{attribute 'linkalways'} 
{attribute 'no_explicit_call' := 'This FB is a CLASS and must be accessed using methods or properties'}
{attribute 'enable_dynamic_creation'}
FUNCTION_BLOCK _ULINT EXTENDS NumericDatatypeBase
VAR
	localData : ULINT;
	activeData : REFERENCE TO ULINT REF= localData;
END_VAR

PROPERTY PUBLIC Address : PVOID
GET
Address := ADR(activeData);
END_GET
END_PROPERTY

METHOD PUBLIC ClearReference
VAR_INPUT
END_VAR
activeData REF= localData;
END_METHOD

METHOD PUBLIC Clone : I_Datatype
VAR
    pClone : POINTER TO _ULINT;
END_VAR
pClone := __NEW(_ULINT(InitialValue := Value));
Clone := pClone^;
END_METHOD

METHOD FB_init : BOOL
VAR_INPUT
	bInitRetains : BOOL; // if TRUE, the retain variables are initialized (warm start / cold start)
	bInCopyCode : BOOL;  // if TRUE, the instance afterwards gets moved into the copy code (online change)
	InitialValue : ULINT;
END_VAR
localData := InitialValue;
END_METHOD

PROPERTY PUBLIC IsFloat : BOOL
GET
IsFloat := FALSE;
END_GET
END_PROPERTY

PROPERTY PUBLIC IsSigned : BOOL
GET
IsSigned := FALSE;
END_GET
END_PROPERTY

PROPERTY PUBLIC LowerBound : ULINT
GET
LowerBound := DatatypeLimits.ULINT_LOWER_LIMIT;
END_GET
END_PROPERTY

METHOD PUBLIC MakeReferenceTo
VAR_INPUT
	ReferenceTarget : REFERENCE TO ULINT;
END_VAR
activeData REF= ReferenceTarget;
END_METHOD

METHOD PROTECTED SerializeLowerbound
VAR_INPUT
	Serializer : I_Serializer;
END_VAR
Serializer.AddUlint(Lowerbound);
END_METHOD

METHOD PROTECTED SerializeUpperbound
VAR_INPUT
	Serializer : I_Serializer;
END_VAR
Serializer.AddUlint(Upperbound);
END_METHOD

METHOD PUBLIC SerializeWith
VAR_INPUT
	Serializer : I_Serializer;
END_VAR
Serializer.AddUlint(activeData);
END_METHOD

PROPERTY PUBLIC Size : UDINT
GET
Size := SIZEOF(activeData);
END_GET
END_PROPERTY

METHOD TryDeserializeFrom : BOOL
VAR_INPUT
	Deserializer : I_Deserializer;
	Feedback : I_DeserializerFeedback;
END_VAR
TryDeserializeFrom := Deserializer.TryGetUlint(activeData, Feedback);
END_METHOD

METHOD TryMakeReferenceTo : BOOL
VAR_INPUT
	Target : I_Datatype;
END_VAR
VAR
	pTargetData : POINTER TO ULINT;
END_VAR
IF NOT (Target.TypeName = TypeName) THEN
	RETURN;
END_IF

pTargetData := Target.Address;
activeData REF= pTargetData^;
TryMakeReferenceTo := TRUE;
END_METHOD

PROPERTY PUBLIC TypeName : T_MAXSTRING
GET
TypeName := 'ULINT';
END_GET
END_PROPERTY

PROPERTY PUBLIC UpperBound : ULINT
GET
UpperBound :=  DatatypeLimits.ULINT_UPPER_LIMIT;
END_GET
END_PROPERTY

PROPERTY PUBLIC Value : ULINT
GET
Value := activeData;
END_GET
SET
activeData := Value;
END_SET
END_PROPERTY

END_FUNCTION_BLOCK

(* stored: Version 1.1.0.1, ProductVersion 3.1.4024.12
   POU _ULINT: Id {ffe5859b-ef46-05bc-36a7-732dc3a25b2e}, SpecialFunc None
   Folder Constructor: Id {e52c06c5-c92b-0354-22f8-1da03a33aaff}
   Folder Protected: Id {015f20a3-2c1b-0965-03ab-ca39ba5df224}
   Property Address: Id {c0e1d138-4876-0997-02d0-e0b39d19c91c}
   Get Get: Id {f24b24fa-8b1a-039a-2a08-2ec4eac8d90d}
   Method ClearReference: Id {03bd0c27-fa0c-0e9d-22e0-4779998be7c7}
   Method Clone: Id {871f4887-9723-0f4d-07a1-2c7c472a1a36}
   Method FB_init: Id {133cedcd-b193-0973-25ad-66022abde12d}
   Property IsFloat: Id {b82c6a2c-69d4-025f-30ca-8009d3c27ddd}
   Get Get: Id {679c90b2-4a4a-08fc-15d3-c56b0ae30d3b}
   Property IsSigned: Id {74ffe30a-6748-09a5-364c-1a5e86ecacc4}
   Get Get: Id {bfd9d2a0-dd04-0573-34d2-37f61f027ecb}
   Property LowerBound: Id {4cc801a2-bdce-0872-06f5-8189ac9a2f92}
   Get Get: Id {ae88aa0e-00ef-07dd-2d59-231dfc894ea1}
   Method MakeReferenceTo: Id {546f53e9-bcfc-0361-1e58-22851df77222}
   Method SerializeLowerbound: Id {79bcb22e-f58f-0039-2612-5ea617ddb3a6}
   Method SerializeUpperbound: Id {d7e7f1c5-73a5-0f16-0fae-7796a6673869}
   Method SerializeWith: Id {ed514a5c-b5e2-0c18-2a8b-21cf4a07fbaa}
   Property Size: Id {8a03cdd9-4bc8-0011-0232-5b3217c6c2fd}
   Get Get: Id {c41f5a6b-548f-0af0-1910-d3ca5c99ca15}
   Method TryDeserializeFrom: Id {8369d3c7-fe9b-0f55-2766-ed3dfa014fa8}
   Method TryMakeReferenceTo: Id {bcf585e1-9fc0-0921-319c-1cdf393a89e1}
   Property TypeName: Id {bfc7bfbf-7e27-0769-0ccb-39e58442f06b}
   Get Get: Id {a7afb3d6-22de-082c-0522-a12ef87c4f0a}
   Property UpperBound: Id {aa968b32-676f-00cb-1c47-19124d0a68e7}
   Get Get: Id {843898d8-4509-0a1c-22f8-9e192b3c2810}
   Property Value: Id {9a36ecbf-09d6-02a0-11b1-c3c15cd2311d}
   Get Get: Id {8184c591-b95d-0ae3-287a-a6a87b75073b}
   Set Set: Id {d3f9b22a-9c1b-0b16-29aa-3c9ca8fb202b} *)
